PROGRAM SavePresistent
VAR
	fbZapisZmiennychPresistent: FB_WritePersistentData;
END_VAR

fbZapisZmiennychPresistent(
	NETID:= , 
	PORT:=851, 
	START:= .bEstopOk OR .bCycleStartCmd OR .bCycleStopCmd OR .bControlOn, 
	TMOUT:=T#2000MS , 
	MODE:=SPDM_2PASS , 
	BUSY=> , 
	ERR=> , 
	ERRID=> );

END_PROGRAM

(* stored: Version 1.1.0.1, ProductVersion 3.1.4024.15
   POU SavePresistent: Id {3d257d62-9ca1-4b9f-9360-0b1ff7a8c3cf}, SpecialFunc None *)
